DATA_BLOCK "ServoV90_A2"
{ S7_Optimized_Access := 'FALSE' }
VERSION : 0.1
NON_RETAIN
// ATTRIBUTES
// AUTO_NUMBER = False
// BLOCK_NUMBER = 2502
// END_ATTRIBUTES
   STRUCT
      In : Struct
         iInterlock : Bool;
         "iManJog+" : Bool;
         "iManJog-" : Bool;
         iAutoStart : Bool;
         iHome : Bool;
         iCancelTask : Bool;
         iPauseTask : Bool;
         iManStart : Bool;
         iManListStart : Bool;
         iLimitSwitchActive : Bool;
         iLimitSoftActive : Bool;
         iRunningTimeout : Time;
         iHomingTimeout : Time;
         iAutoPosition : DInt;
         iAutoVelocity : Int;
         iManListPosition : DInt;
         iManListVelocity : Int;
         iManListNumber : Int;
         iManPosition : DInt;
         iManVelocity : Int;
         iMode : Int;
      END_STRUCT;
      Out : Struct
         oReady : Bool;
         oWarning : Bool;
         oError : Bool;
         oInterlock : Bool;
         oServoEnable : Bool;
         oRunning : Bool;
         oHoming : Bool;
         oHomeRef : Bool;
         oServoPosOK : Bool;
         oErrorCode : Int;
         oStatus : Int;
         oActPosition : DInt;
         oManualListPos : DInt;
      END_STRUCT;
      IO : Struct
         ioManEnale : Bool;
         ioAutoEnale : Bool;
      END_STRUCT;
      Spare : Struct
         S : Array[0..100] of Byte;
      END_STRUCT;
      Manual : Struct
         Index : Int;
         Pos : Array[1..20] of Struct
            Pos : DInt;
            Vel : Int;
         END_STRUCT;
      END_STRUCT;
      Auto : Struct
         Index : Int;
         Pos : Array[1..20] of Struct
            Pos : DInt;
            Vel : Int;
         END_STRUCT;
      END_STRUCT;
      Interlock : Struct
         Active : Bool;
         Case1 : Bool;
         Case2 : Bool;
         Case3 : Bool;
         Case4 : Bool;
         Case5 : Bool;
         Case6 : Bool;
         Case7 : Bool;
         Case8 : Bool;
         Case9 : Bool;
         Case10 : Bool;
      END_STRUCT;
      PositionOk : Array[1..20] of Bool;
      Home_Pos : Struct
         "Home Pos Pls" : Bool;
         "Arrow indication" : Int;
         "Process prompt" : Int;
         "Button prompt" : Int;
      END_STRUCT;
   END_STRUCT;


BEGIN
   In.iInterlock := TRUE;
   In."iManJog+" := FALSE;
   In."iManJog-" := FALSE;
   In.iAutoStart := FALSE;
   In.iHome := FALSE;
   In.iCancelTask := FALSE;
   In.iPauseTask := FALSE;
   In.iManStart := FALSE;
   In.iManListStart := FALSE;
   In.iLimitSwitchActive := TRUE;
   In.iLimitSoftActive := TRUE;
   In.iRunningTimeout := T#0MS;
   In.iHomingTimeout := T#0MS;
   In.iAutoPosition := 0;
   In.iAutoVelocity := 0;
   In.iManListPosition := 0;
   In.iManListVelocity := 0;
   In.iManListNumber := 0;
   In.iManPosition := 0;
   In.iManVelocity := 0;
   In.iMode := 0;
   Out.oReady := FALSE;
   Out.oWarning := FALSE;
   Out.oError := TRUE;
   Out.oInterlock := TRUE;
   Out.oServoEnable := FALSE;
   Out.oRunning := FALSE;
   Out.oHoming := FALSE;
   Out.oHomeRef := TRUE;
   Out.oServoPosOK := FALSE;
   Out.oErrorCode := -244;
   Out.oStatus := 0;
   Out.oActPosition := 113;
   Out.oManualListPos := 0;
   IO.ioManEnale := FALSE;
   IO.ioAutoEnale := FALSE;
   Spare.S[0] := 16#00;
   Spare.S[1] := 16#00;
   Spare.S[2] := 16#00;
   Spare.S[3] := 16#00;
   Spare.S[4] := 16#00;
   Spare.S[5] := 16#00;
   Spare.S[6] := 16#00;
   Spare.S[7] := 16#00;
   Spare.S[8] := 16#00;
   Spare.S[9] := 16#00;
   Spare.S[10] := 16#00;
   Spare.S[11] := 16#00;
   Spare.S[12] := 16#00;
   Spare.S[13] := 16#00;
   Spare.S[14] := 16#00;
   Spare.S[15] := 16#00;
   Spare.S[16] := 16#00;
   Spare.S[17] := 16#00;
   Spare.S[18] := 16#00;
   Spare.S[19] := 16#00;
   Spare.S[20] := 16#00;
   Spare.S[21] := 16#00;
   Spare.S[22] := 16#00;
   Spare.S[23] := 16#00;
   Spare.S[24] := 16#00;
   Spare.S[25] := 16#00;
   Spare.S[26] := 16#00;
   Spare.S[27] := 16#00;
   Spare.S[28] := 16#00;
   Spare.S[29] := 16#00;
   Spare.S[30] := 16#00;
   Spare.S[31] := 16#00;
   Spare.S[32] := 16#00;
   Spare.S[33] := 16#00;
   Spare.S[34] := 16#00;
   Spare.S[35] := 16#00;
   Spare.S[36] := 16#00;
   Spare.S[37] := 16#00;
   Spare.S[38] := 16#00;
   Spare.S[39] := 16#00;
   Spare.S[40] := 16#00;
   Spare.S[41] := 16#00;
   Spare.S[42] := 16#00;
   Spare.S[43] := 16#00;
   Spare.S[44] := 16#00;
   Spare.S[45] := 16#00;
   Spare.S[46] := 16#00;
   Spare.S[47] := 16#00;
   Spare.S[48] := 16#00;
   Spare.S[49] := 16#00;
   Spare.S[50] := 16#00;
   Spare.S[51] := 16#00;
   Spare.S[52] := 16#00;
   Spare.S[53] := 16#00;
   Spare.S[54] := 16#00;
   Spare.S[55] := 16#00;
   Spare.S[56] := 16#00;
   Spare.S[57] := 16#00;
   Spare.S[58] := 16#00;
   Spare.S[59] := 16#00;
   Spare.S[60] := 16#00;
   Spare.S[61] := 16#00;
   Spare.S[62] := 16#00;
   Spare.S[63] := 16#00;
   Spare.S[64] := 16#00;
   Spare.S[65] := 16#00;
   Spare.S[66] := 16#00;
   Spare.S[67] := 16#00;
   Spare.S[68] := 16#00;
   Spare.S[69] := 16#00;
   Spare.S[70] := 16#00;
   Spare.S[71] := 16#00;
   Spare.S[72] := 16#00;
   Spare.S[73] := 16#00;
   Spare.S[74] := 16#00;
   Spare.S[75] := 16#00;
   Spare.S[76] := 16#00;
   Spare.S[77] := 16#00;
   Spare.S[78] := 16#00;
   Spare.S[79] := 16#00;
   Spare.S[80] := 16#00;
   Spare.S[81] := 16#00;
   Spare.S[82] := 16#00;
   Spare.S[83] := 16#00;
   Spare.S[84] := 16#00;
   Spare.S[85] := 16#00;
   Spare.S[86] := 16#00;
   Spare.S[87] := 16#00;
   Spare.S[88] := 16#00;
   Spare.S[89] := 16#00;
   Spare.S[90] := 16#00;
   Spare.S[91] := 16#00;
   Spare.S[92] := 16#00;
   Spare.S[93] := 16#00;
   Spare.S[94] := 16#00;
   Spare.S[95] := 16#00;
   Spare.S[96] := 16#00;
   Spare.S[97] := 16#00;
   Spare.S[98] := 16#00;
   Spare.S[99] := 16#00;
   Spare.S[100] := 16#00;
   Manual.Index := 1;
   Manual.Pos[1].Pos := 0;
   Manual.Pos[1].Vel := 10000;
   Manual.Pos[2].Pos := 450000;
   Manual.Pos[2].Vel := 10000;
   Manual.Pos[3].Pos := 900000;
   Manual.Pos[3].Vel := 10000;
   Manual.Pos[4].Pos := 135000;
   Manual.Pos[4].Vel := 10000;
   Manual.Pos[5].Pos := 180000;
   Manual.Pos[5].Vel := 10000;
   Manual.Pos[6].Pos := 225000;
   Manual.Pos[6].Vel := 10000;
   Manual.Pos[7].Pos := 270000;
   Manual.Pos[7].Vel := 10000;
   Manual.Pos[8].Pos := 315000;
   Manual.Pos[8].Vel := 10000;
   Manual.Pos[9].Pos := 0;
   Manual.Pos[9].Vel := 0;
   Manual.Pos[10].Pos := 0;
   Manual.Pos[10].Vel := 0;
   Manual.Pos[11].Pos := 0;
   Manual.Pos[11].Vel := 0;
   Manual.Pos[12].Pos := 0;
   Manual.Pos[12].Vel := 0;
   Manual.Pos[13].Pos := 0;
   Manual.Pos[13].Vel := 0;
   Manual.Pos[14].Pos := 0;
   Manual.Pos[14].Vel := 0;
   Manual.Pos[15].Pos := 0;
   Manual.Pos[15].Vel := 0;
   Manual.Pos[16].Pos := 0;
   Manual.Pos[16].Vel := 0;
   Manual.Pos[17].Pos := 0;
   Manual.Pos[17].Vel := 0;
   Manual.Pos[18].Pos := 0;
   Manual.Pos[18].Vel := 0;
   Manual.Pos[19].Pos := 0;
   Manual.Pos[19].Vel := 0;
   Manual.Pos[20].Pos := 0;
   Manual.Pos[20].Vel := 0;
   Auto.Index := 1;
   Auto.Pos[1].Pos := 0;
   Auto.Pos[1].Vel := 10000;
   Auto.Pos[2].Pos := 450000;
   Auto.Pos[2].Vel := 10000;
   Auto.Pos[3].Pos := 900000;
   Auto.Pos[3].Vel := 10000;
   Auto.Pos[4].Pos := 135000;
   Auto.Pos[4].Vel := 10000;
   Auto.Pos[5].Pos := 180000;
   Auto.Pos[5].Vel := 10000;
   Auto.Pos[6].Pos := 225000;
   Auto.Pos[6].Vel := 10000;
   Auto.Pos[7].Pos := 270000;
   Auto.Pos[7].Vel := 10000;
   Auto.Pos[8].Pos := 315000;
   Auto.Pos[8].Vel := 10000;
   Auto.Pos[9].Pos := 0;
   Auto.Pos[9].Vel := 0;
   Auto.Pos[10].Pos := 0;
   Auto.Pos[10].Vel := 0;
   Auto.Pos[11].Pos := 0;
   Auto.Pos[11].Vel := 0;
   Auto.Pos[12].Pos := 0;
   Auto.Pos[12].Vel := 0;
   Auto.Pos[13].Pos := 0;
   Auto.Pos[13].Vel := 0;
   Auto.Pos[14].Pos := 0;
   Auto.Pos[14].Vel := 0;
   Auto.Pos[15].Pos := 0;
   Auto.Pos[15].Vel := 0;
   Auto.Pos[16].Pos := 0;
   Auto.Pos[16].Vel := 0;
   Auto.Pos[17].Pos := 0;
   Auto.Pos[17].Vel := 0;
   Auto.Pos[18].Pos := 0;
   Auto.Pos[18].Vel := 0;
   Auto.Pos[19].Pos := 0;
   Auto.Pos[19].Vel := 0;
   Auto.Pos[20].Pos := 0;
   Auto.Pos[20].Vel := 0;
   Interlock.Active := FALSE;
   Interlock.Case1 := TRUE;
   Interlock.Case2 := TRUE;
   Interlock.Case3 := FALSE;
   Interlock.Case4 := FALSE;
   Interlock.Case5 := FALSE;
   Interlock.Case6 := FALSE;
   Interlock.Case7 := FALSE;
   Interlock.Case8 := FALSE;
   Interlock.Case9 := FALSE;
   Interlock.Case10 := FALSE;
   PositionOk[1] := FALSE;
   PositionOk[2] := FALSE;
   PositionOk[3] := FALSE;
   PositionOk[4] := FALSE;
   PositionOk[5] := FALSE;
   PositionOk[6] := FALSE;
   PositionOk[7] := FALSE;
   PositionOk[8] := FALSE;
   PositionOk[9] := FALSE;
   PositionOk[10] := FALSE;
   PositionOk[11] := FALSE;
   PositionOk[12] := FALSE;
   PositionOk[13] := FALSE;
   PositionOk[14] := FALSE;
   PositionOk[15] := FALSE;
   PositionOk[16] := FALSE;
   PositionOk[17] := FALSE;
   PositionOk[18] := FALSE;
   PositionOk[19] := FALSE;
   PositionOk[20] := FALSE;
   Home_Pos."Home Pos Pls" := FALSE;
   Home_Pos."Arrow indication" := 0;
   Home_Pos."Process prompt" := 0;
   Home_Pos."Button prompt" := 0;

END_DATA_BLOCK

